{attribute 'linkalways'} 
{attribute 'no_explicit_call' := 'This FB is a CLASS and must be accessed using methods or properties'}
{attribute 'enable_dynamic_creation'}
FUNCTION_BLOCK Node_ContainerType_Vector_UINT EXTENDS Node
VAR
    out : _GUID;
END_VAR

METHOD PUBLIC  Clone : I_Node
VAR
	pNode : POINTER TO Node_ContainerType_Vector_UINT;
END_VAR
pNode := __NEW(Node_ContainerType_Vector_UINT);
Clone := pNode^;
END_METHOD

METHOD FB_init : BOOL
VAR_INPUT
	bInitRetains : BOOL; // if TRUE, the retain variables are initialized (warm start / cold start)
	bInCopyCode : BOOL;  // if TRUE, the instance afterwards gets moved into the copy code (online change)
END_VAR
AddOutput('out', out);
END_METHOD

METHOD PROTECTED OnExecute
out.Value := ContainerType_Vector_UINT;
END_METHOD

END_FUNCTION_BLOCK

(* stored: Version 1.1.0.1, ProductVersion 3.1.4026.17
   POU Node_ContainerType_Vector_UINT: Id {e4de2151-2f3e-0b30-0ada-40e992315cf8}, SpecialFunc None
   Folder Constructor: Id {a04dbd5d-7567-055f-2fdd-1dce5eeec6fd}
   Method Clone: Id {9fa8132e-5dd3-0920-1cad-1ca290045134}
   Method FB_init: Id {ebacb533-b1d0-0a68-21ce-2fe07e711384}
   Method OnExecute: Id {3878baf1-ac06-0aea-1112-418a68183964} *)
